Staubli VAL3: ImpedCtrlTest.pjx

--- ImpedCtrlTest.pjx ---
Parameters version=s7.9.1 stackSize=50000 millimeterUnit=true
Program file=ASCIItoNum.pgx
Program file=calcForce.pgx
Program file=dataUpdate.pgx
Program file=errorCalc.pgx
Program file=initSensor.pgx
Program file=loopReadForce.pgx
Program file=newCommand.pgx
Program file=readDeteVal.pgx
Program file=start.pgx
Program file=stop.pgx
Program file=userInterface.pgx
Data file=ImpedCtrlTest.dtx

--- ImpedCtrlTest.dtx ---
mdesc mNomSpeed
public bool bOverRun = true
public num nMass[6 6]
  [0,0] = 1
  [1,1] = 1
  [2,2] = 1
  [3,3] = 1
  [4,4] = 1
  [5,5] = 1
public num nStiffness[6 6]
  [0,0] = 25
  [1,1] = 25
  [2,2] = 25
  [3,3] = 25
  [4,4] = 25
  [5,5] = 25
public num nDamp[6 6]
  [0,0] = 10
  [1,1] = 10
  [2,2] = 10
  [3,3] = 10
  [4,4] = 10
  [5,5] = 10
public num ndForce[6]
public num ndAccel[6]
public num ndVelocity[6]
public num nForce[6]
public num ndPosition[6]
public mdesc mImpedSpeed = {blend=off}
public pointRx pNowPosition = {fatherId=world[0]}
public num nNowVelocity[6]
public num nNowAccel[6]
public num nLastVelocity[6]
public num nNowClock
public num nTime
public sio sClient = {link=Socket\FTSensor}
public num nForceTorque[6]
  [0] = -0.458435
  [1] = -0.0611247
  [2] = -0.0305157
  [3] = 0.00182448
  [4] = 0.00243784
public num nPort = 5001
public num nSensitivity[6]
  [0] = 32.72
  [1] = 32.72
  [2] = 32.77
  [3] = 1644.3
  [4] = 1640.8
  [5] = 1635
public num nSioTimeOut = 5
public num nZeroPoint[6]
  [0] = 8211
  [1] = 8189
  [2] = 8176
  [3] = 8194
  [4] = 8176
  [5] = 8189
public pointRx pCommand = {fatherId=world[0]}

--- start.pgx ---
program start()
  local bool l_bActive
  local jointRx l_jInitPoint
  local jointRx l_jStartPoint
  local string l_sConnect
begin

  //--------------------WACOH F/T Sensor的操作力/力矩信息采集、过滤及传输显示---------------------
  //初始化Wacoh Force/Torque Sensor
  call initSensor("io:Wacoh",l_sConnect)
  if l_sConnect=="yes"
    putln("Connection success!")
    delay(1)
  else
    putln("Connection fail!")
    delay(1)
  endIf

  //创建同步任务，循环获取传感器的Force/Torque数据（采集频率0.004s，频率为250Hz，可设置调节，超时是否需打开？）
  taskCreateSync "getForces",0.004,bOverRun,loopReadForce()

  //创建异步任务，将采集的传感器数据发送至用户界面实时显示
  taskCreate "user",100,userInterface()



  //---------------------机器人Staubli运动控制---------------------
  //机器人复位（回到默认初始关节角均为0的状态）
  l_jInitPoint={50,40,75,0,65,0}
  resetMotion(l_jInitPoint)
  autoConnectMove(l_bActive)

  //移动至开始运动点
  l_jStartPoint={60,40,75,0,65,0}
  movej(l_jStartPoint,flange,mNomSpeed)
  waitEndMove()


  //设定机器人的初始状态（假设初始速度和加速度均为0），用于生成机器人的第一次运动指令----------
  pNowPosition=$getPosFbk(flange,world)
  nLastVelocity=0
  nNowVelocity=0
  nNowAccel=0
  nNowClock=clock()
  //第一次定义执行时间
  nTime=0.004

  //更新机器人数据、计算并执行新的指令、获取当前的机器人状态（位置、速度、加速度），为下一个机器人运动指令做好准备----------
  //创建同步任务更新数据（Sensor力/力矩，参考力，参考运动，阻抗参数）
  taskCreateSync "dataUpdate",0.004,bOverRun,dataUpdate(nForceTorque)

  //创建异步位置更新并执行位置指令
  taskCreate "newCommand",100,newCommand()

end

--- errorCalc.pgx ---
public program errorCalc(pointRx& x_pNewPostion[])
  local num l_nAccel[6]
  local num l_nNewPosition[6]
  local num l_nNowPosition[6]
  local num l_nNum
  local num l_nTime
  local num l_nVelocity[6]
  local pointRx l_pNowPosTemp
  local pointRx l_pPosTemp
begin

  //计算机器人指令误差，并生成新的位置---------
  //获取机器人执行运动指令时间
  l_nTime=nTime

  //将机器人的当前位置赋值给数组变量，便于程序操作
  l_pPosTemp=pNowPosition
  l_nNowPosition[0]=l_pPosTemp.trsf.x
  l_nNowPosition[1]=l_pPosTemp.trsf.y
  l_nNowPosition[2]=l_pPosTemp.trsf.z
  l_nNowPosition[3]=l_pPosTemp.trsf.rx
  l_nNowPosition[4]=l_pPosTemp.trsf.ry
  l_nNowPosition[5]=l_pPosTemp.trsf.rz

  //求加速度（位置+姿态）
  for l_nNum=0 to 5
    l_nAccel[l_nNum]=ndAccel[l_nNum]+1/nMass[l_nNum,l_nNum]*(-(ndForce[l_nNum]-nForce[l_nNum])-nDamp[l_nNum,l_nNum]/1000*(nNowVelocity[l_nNum]-ndVelocity[l_nNum])-nStiffness[l_nNum,l_nNum]/1000*(l_nNowPosition[l_nNum]-ndPosition[l_nNum]))
  endFor

  //求速度（位置+姿态）
  for l_nNum=0 to 5
    l_nVelocity[l_nNum]=nNowVelocity[l_nNum]/1000+l_nAccel[l_nNum]*l_nTime
  endFor

  //求位置指令（位置+姿态）（转换成笛卡儿坐标点类型）
  for l_nNum=0 to 5
    l_nNewPosition[l_nNum]=l_nNowPosition[l_nNum]+l_nVelocity[l_nNum]*1000*l_nTime
  endFor
  x_pNewPostion.trsf.x=l_nNewPosition[0]
  x_pNewPostion.trsf.y=l_nNewPosition[1]
  x_pNewPostion.trsf.z=l_nNewPosition[2]
//  x_pNewPostion.trsf.rx=l_nNewPosition[3]/60
//  x_pNewPostion.trsf.ry=l_nNewPosition[4]/60
//  x_pNewPostion.trsf.rz=l_nNewPosition[5]/60
  x_pNewPostion.trsf.rx=0
  x_pNewPostion.trsf.ry=-180
  x_pNewPostion.trsf.rz=-60
  delay(0)

end

--- loopReadForce.pgx ---
public program loopReadForce()
  local num l_nDetectValue[6]
begin

  //循环调用函数readDetectValue()读取传感器数值并转换成Force/Torque值------------
  do
    //获取传感器的当前检测值
    call readDeteVal(l_nDetectValue)

    //计算传感器的Force/Torque数值并输出
    call calcForce(l_nDetectValue,nForceTorque)
    delay(0)

  until false

end

--- newCommand.pgx ---
public program newCommand()
  local num l_nNum
  local num l_nNowClock
  local num l_nLastClock
  local num l_nTime
  local pointRx l_pCommand
begin

  //循环生成并执行新的机器人位置指令且记录当前机器人的状态（可在此时运行同步任务获取机器人状态）
  do
    //计算机器人新的位置指令----------
    call errorCalc(pCommand)


    //执行新的位置指令-----------
    alterMovej(pCommand,flange,mImpedSpeed)
    //waitEndMove()


    //获取时钟状态并计算movej指令执行时间----------
    l_nLastClock=nNowClock
    nNowClock=clock()
    l_nNowClock=nNowClock
    l_nTime=l_nNowClock-l_nLastClock
    nTime=l_nTime


    //获取机器人当前的状态（位置，速度，加速度）----------
    //获取机器人的当前位置，并赋值给数组变量，便于程序操作（作为下一条指令计算中的当前位置）
    pNowPosition=$getPosFbk(flange,world)

    //获取机器人的前一次及当前笛卡尔速度（有待考证和计算）
    //nLastVelocity=nNowVelocity
    for l_nNum= 0 to 5
      nLastVelocity[l_nNum]=nNowVelocity[l_nNum]
    endFor
    $getSpeedFbk(flange,world,nNowVelocity[0],nNowVelocity[1],nNowVelocity[2],nNowVelocity[3],nNowVelocity[4],nNowVelocity[5])

    //计算机器人的当前加速度（位置+姿态）（利用当前和上一个速度差分计算）
//    for l_nNum= 0 to 5
//      nNowAccel[l_nNum]=(nNowVelocity[l_nNum]-nLastVelocity[l_nNum])/l_nTime
//    endFor

    delay(0.0)

  until false

end

--- stop.pgx ---
program stop()
begin

  //test command

end
